PROGRAM P_Gang_5_153D
VAR

	fbLys		: FB_Light_Type_B;
	

	stDaliSetup	: SH_Light.ST_DALI_RoomSetup := (
														byShrtAdr_Prim := 47, 
														byGrpAdr_Prim := 10, 
														eMod_Prim := E_DALIAddressType.Group, 
														//byShrtAdr_Sec := 1, 
														//byGrpAdr_Sec := 1, 
														//eMod_Sec := E_DALIAddressType.Short, 
														//byShrtAdr_Supl := 1,
														//byGrpAdr_Supl := 1,
														//eMod_Prim := E_DALIAddressType.Short
														DALI_LINE_NUM_PRIM := DALI_LINE_NUM_LIGHT, 
														DALI_LINE_NUM_SEC := 0, //0 = ingen zonestyring/vinduerække
														DALI_LINE_NUM_SUPL := DALI_LINE_NUM_PENDANTS);
														
	stLiveData					: SH_Light.ST_LiveData;
	bRunTuning					: BOOL;
	
	bTopButtonZone1			: BOOL;
	bTopButtonZone1_Visu	: BOOL;
	bBottomButtonZone1		: BOOL;
	bBottomButtonZone1_Visu	: BOOL;
	bButtonZone2				: BOOL;
	bNeighborRoomsPir		: BOOL;
	fLuxOn							: REAL;
	fLuxDim						: REAL;
	tPIRDim						: TIME;
	tPIROff						: TIME;
	fOffsetSec					: REAL := 20;
	bOccupiedRoom			: BOOL;


// Sensor Settings
	fbSensor						: SH_Light.FB_NIKO_P46xx_1Pcs;
	//fbSensor						: SH_Light.FB_NIKO_P46xx_3Pcs;
	bySensorAddr				: BYTE := 3;
	//arrSensorAddr				: ARRAY[1..3] OF BYTE := [7,8,9];
	bInitialize						: BOOL := TRUE;
	stDaliSensorSetup			: ST_DALI_NIKOP46SetupData := (
																nSensitivityPIRSegmentA := arrSensitivityOccupancy[1],
																nSensitivityPIRSegmentB := arrSensitivityOccupancy[2],
																nSensitivityPIRSegmentC := arrSensitivityOccupancy[3]);
//	arrSensitivityOccupancy				: ARRAY[1..3] OF BYTE := [4,4,4];
	bInitErr							: BOOL;
	bInitDone						: BOOL;
	//arrInitErr						: ARRAY [1..3] OF BOOL;
	//arrInitDone					: ARRAY [1..3] OF BOOL;
	arrSensorScales				: ARRAY [1..10] OF SH_Light.ST_DALI_SensorScaleMode := [
																						(fMeassureMaxSensor := rMeassure_Zone5, fReadMaxSensor := rRead_Zone5),																																										
																						9(())];
	bCancelHoldTimerOccupancy	: BOOL;
(*	eEventPriorityOccupancy		: E_DALIEventPriority := E_DALIEVENTPRIORITY.Middle;
	nHoldTimerOccupancy			: WORD := 5; // Value in s. 	
	nReportTimerOccupancy		: BYTE := 120; // Value in s, Preset manufacturer value
	nDeadtimeTimerOccupancy		: WORD := 100; // Value in ms, Predefined Value of DALI Standard
	bCancelHoldTimerOccupancy	: BOOL;
	nSensitivityOccupancy		: BYTE:= 3; //setting Sensivity (0..4) 0 (Off), 1 (Min), 2(Low), 3(High) and 4 (Max)

	bEnableLuxEvent				: BOOL;
	eEventPriorityBrightness	: E_DALIEventPriority := E_DALIEVENTPRIORITY.Middle;
	nDeadtimeTimerBrightness	: WORD := 1500; // Value in ms, Predefined Value of DALI Standard
	nHysteresisBrightness		: BYTE := 2; // Value in %
	nHysteresisMinBrightness	: BYTE := 10; // Absolute Value, depending on the manufacturer specific resolution
	nReportTimerBrightness		: BYTE := 120; // Value in s, Preset manufacturer value
*)

	//stDaliSetup: SH_Light.ST_DALI_RoomSetup
	//stRoomDataModbus			: SH_Light.ST_RoomDataModbus := ( bPirActive := bPirActive
	

	//ModbusComm setup
	
	fbWriteSPLuxLevel			: SH_Light.FB_TwoVal_SelectOne_RTrigChange;
	fbWritePirDelayTIme		: SH_Light.FB_TwoVal_SelectOne_RTrigChange;
	stRoomDataPLC				: SH_Light.ST_RoomDataPLC	:=	(
																	uiPirOffDelayTime	:= 30,
																	uiSpLuxLevel			:= 500,
																	uiPirDimDelayTime	:= 15,
																	uiSpDimLuxLevel		:= 200);
																	
	fbBallastOnHours				: SH_Light.FB_CountOnHours;
	bEnableHourCount			: BOOL := TRUE;
	
	//Non-persistent modbus data
	bPirActive_MB					AT %MX116.0	: BOOL;				//bPirLys i gammel kode
	uiActLuxLevel_MB			AT %MB120	: UINT;				//intHMIAktueltLux i gammel kode
	uiActLightLevelPct_MB	AT %MB124	: UINT;				//intDALI_Gruppe1_Lysniveau i gammel kode
	
	//For Conversion
	uiPirOffMinutes						: UINT;
	udTimeScaling						: UDINT := 60000;
	uiLuxOn								: UINT;
	
	//max values checks
	uiMaxLuxLevel						: UINT := 1023;
	uiMaxPirOffMinutes				: UINT := 180;

	
END_VAR

VAR CONSTANT
    Sensor_DALI_LINE_NUM				: BYTE := 3;
	DALI_LINE_NUM_LIGHT				: BYTE := 1;
	DALI_LINE_NUM_PENDANTS	: BYTE := 0; //0=ingen pendler	
	arrSensitivityOccupancy				: ARRAY[1..3] OF BYTE := [4,4,4];
END_VAR
VAR PERSISTENT
	stPirSensorData: SH_Light.ST_DALI_Sensor;
	stTuneData: SH_Light.ST_TuneData_EX;

	uiPirOffDelayTime_MB		AT %MB118	: UINT;				//ntHMI_Pir_SetValue i gammel kode
	uiSPLuxLevel_MB			AT %MB122	: UINT;				//intHMI_Lux_SetValue i gammel kode
	uiBallastOnHours_MB		AT %MB126	: UINT;				//dintHMILysbraendtimer1 i gammel kode
	byOnHoursOverflowCount							: BYTE;   
END_VAR

A_Buttons();
A_LightCtrl();
A_Sensor();
A_ModbusComm();

ACTION A_Buttons:
bTopButtonZone1		:= GVL_EnOcean.strEnOceanSwitch_Gang_5_153D.bT2_ON OR bTopButtonZone1_Visu;
bBottomButtonZone1	:= GVL_EnOcean.strEnOceanSwitch_Gang_5_153D.bT2_OFF OR  bBottomButtonZone1_Visu;
END_ACTION

ACTION A_LightCtrl:
bNeighborRoomsPir :=	P_Gang_5_153A.stPirSensorData.bPrc OR
									P_Gang_5_153C.stPirSensorData.bPrc ;
fbLys(
	nZoneID:= 1, 
	bButtonZone1:= bTopButtonZone1,
	bBottomButtonZone1 := bBottomButtonZone1, 
	//bButtonZone2:= bButtonZone2,
	bNeighborRoomsPir := bNeighborRoomsPir,
	fLuxOn:= fLuxOn, 
	fLuxDim:= fLuxDim, 
	tPIRDim:= tPIRDim, 
	tPIROff:= tPIROff, 
	fOffsetSec:= fOffsetSec, 
	bReInit:= , 
	stDaliSetup:= stDaliSetup, 
	ipCommunication_Prim:= P_DALI_Background.arrfbKL6821Communication[DALI_LINE_NUM_LIGHT], 
	//ipCommunication_Sec:= P_DALI_Background.arrfbKL6821Communication[DALI_LINE_NUM_LIGHT], 
	//ipCommunication_Supl:= P_DALI_Background.arrfbKL6821Communication[DALI_LINE_NUM_PENDANTS], 
	fMinOutputPowerLevelRoom:= 15, 
	fMaxOutputPowerLevelRoom:= 100, 
	nCycleTimeInMS:= SH_Light.DALI_Param.nPlcTaskCycleTimeInMS*nDimCmdCycleTimeFactor , 
	bRunTuning:= bRunTuning, 
	bOccupiedRoom=> bOccupiedRoom, 
	bError_Prim=> , 
	nError_Prim=> , 
	stTuneData:=stTuneData , 
	stPirSensorData:= stPirSensorData, 
	stLiveData:= stLiveData);
END_ACTION

ACTION A_ModbusComm:
//Manage data for modbus communication

//Manage data for read-only in PLC
stRoomDataPLC.bPirActive			:= stPirSensorData.bPrc;
stRoomDataPLC.uiActLuxLevel			:= TO_UINT(TRUNC(stPirSensorData.fBrightness));
stRoomDataPLC.uiActLightLevelPct	:= TO_UINT(TRUNC(fbLys.fbBallast.fActlLgtLvl_Prim));
		//stRoomDataPLC.uiActLightLevelPct	:= TO_UINT(TRUNC(fbLys.fbBallast.fActlLgtLvl_Prim)); //if only one group light control
stRoomDataPLC.uiBallastOnHours		:= uiBallastOnHours_MB; //The calculation for BallastOnHours is stored directly to the MB register below


//Assign data for read-only to MB registers
bPirActive_MB			:= stRoomDataPLC.bPirActive;
uiActLuxLevel_MB		:= stRoomDataPLC.uiActLuxLevel;
uiActLightLevelPct_MB	:= stRoomDataPLC.uiActLightLevelPct;

	//calculate BallastOnHours
	fbBallastOnHours(
		bEnableHourCount	:= bEnableHourCount,
		bPauseCount			:= fbLys.fbLightCtrl.bOffZone1,
		uiOnHours			:= uiBallastOnHours_MB,			//OnHours is updated here
		byOverflowCount		:= byOnHoursOverflowCount);


//Manage data for read/write for both PLC and MB registers
fbWriteSPLuxLevel(	nMaxValOut	:= uiMaxLuxLevel,
					nValIn1		:= uiSPLuxLevel_MB,		//nValIn1 takes priotity in case of download or restart
					nValIn2		:= stRoomDataPLC.uiSpLuxLevel,
					nValOut		=> uiLuxOn
				);


fbWritePirDelayTIme(	nMaxValOut	:= uiMaxPirOffMinutes,
						nValIn1		:= uiPirOffDelayTime_MB,		//nValIn1 takes priotity in case of download or restart
						nValIn2		:= stRoomDataPLC.uiPirOffDelayTime,
						nValOut		=> uiPirOffMinutes
					);
					

//Convert read/write modbus data to appropriate datatypes in PLC
fLuxOn	:= TO_REAL(uiLuxOn);			
tPIROff	:= TO_TIME(uiPirOffMinutes*udTimeScaling); //Time conversion defaults to ms

fLuxDim	:= TO_REAL(stRoomDataPLC.uiSpDimLuxLevel);			
tPIRDim	:= TO_TIME(stRoomDataPLC.uiPirDimDelayTime*udTimeScaling); //Time conversion defaults to ms
END_ACTION

ACTION A_Sensor:

fbSensor.ipCommunication := P_DALI_Background.arrfbKL6821Communication[Sensor_DALI_LINE_NUM];

//only 1 sensor
fbSensor(
	byShrtAdr:= bySensorAddr,
	bInitialize:= bInitialize, 
	DALI_LINE_NUM:= Sensor_DALI_LINE_NUM, 
 	//bCancelHoldTimerOccupancy:= bCancelHoldTimerOccupancy, 
	stSensorSetup := stDaliSensorSetup,
	bInitErr=> bInitErr, 
	bInitDone=> bInitDone,
	stPirSensorData:= stPirSensorData, 
	arrSensorScales:= arrSensorScales);


(*//several sensors	
fbSensor(
	arrShrtAdr:= arrSensorAddr,
	bInitialize:= bInitialize, 
	DALI_LINE_NUM:= Sensor_DALI_LINE_NUM, 
 	//bCancelHoldTimerOccupancy:= bCancelHoldTimerOccupancy, 
	stSensorSetup := stDaliSensorSetup,
	arrInitErr=> arrInitErr, 
	arrInitDone=> arrInitDone,
	stPirSensorData:= stPirSensorData, 
	arrSensorScales:= arrSensorScales);
	*)
END_ACTION

END_PROGRAM

(* stored: Version 1.1.0.1
   POU P_Gang_5_153D: Id {ec0f4b3c-1042-4514-8e36-71ef69a33b19}, SpecialFunc None
   Action A_Buttons: Id {48209050-5f57-4bfd-9451-a991ca27925c}
   Action A_LightCtrl: Id {fd059a7c-dfae-48ad-86da-6b4b08fd247b}
   Action A_ModbusComm: Id {378017b3-09e0-43bd-9a10-23befe4eba50}
   Action A_Sensor: Id {06046676-0c6d-43cd-baf1-84fa40ea3896} *)
